// TwinCAT 3 PLC project Untitled1
// ProgramVersion: 3.1.4023.0
// libraries:
//   Tc2_Standard, * (Beckhoff Automation GmbH)
//   Tc2_System, * (Beckhoff Automation GmbH)
//   Tc3_Module, * (Beckhoff Automation GmbH)
// project tree:
//   DataProcessing/QuickSort/ Partition.TcPOU, QuickSort.TcPOU, Swap.TcPOU
//   GVLs/ GVL.TcGVL
//   List/ ListOfINT.TcPOU, NodeINT.TcDUT (not stored)
//   / PlcTask.TcTTO
//   POUs/ ListOfINTTest.TcPOU, MAIN.TcPOU, QuickSortTest.TcPOU
//   Stringify/ Stringify.TcPOU

CONFIGURATION Untitled1
    RESOURCE PLC ON TwinCAT3
        TASK PlcTask(INTERVAL := T#10ms, PRIORITY := 20);
        PROGRAM MAIN WITH PlcTask : MAIN;
    END_RESOURCE
END_CONFIGURATION

// ---- GVLs/GVL.TcGVL
{attribute 'qualified_only'}
VAR_GLOBAL
	vari : int;
END_VAR

// ---- POUs/MAIN.TcPOU

PROGRAM MAIN
VAR
	
END_VAR


ListOfINTTest();

QuickSortTest();

END_PROGRAM

// ---- POUs/ListOfINTTest.TcPOU
PROGRAM ListOfINTTest
VAR
	listOfINTExample : ListOfINT;
	
	// init
	first : BOOL := TRUE;
	reinit : BOOL;
	
	// insert test
	insertTest : BOOL;
	insertNumber : INT := 42;
	insertIndex : INT := 0;
	
	// remove test
	removeTest : BOOL;
	removeIndex : INT := 0;
	
	// prepend test
	prependTest : BOOL;
	prependData : INT := -10;
	
	// removeAll test
	removeAllTest : BOOL;
	
	// debug
	test : ARRAY[0..30] OF INT;
	
	// hokusy pokusy
	info : __SYSTEM.VAR_INFO;
	
END_VAR

IF first THEN
	first := FALSE;
	listOfINTExample.Append(3);
	listOfINTExample.Append(4);
//	listOfINTExample.Append(5).Prepend(2).Prepend(1);
END_IF;
IF reinit THEN
	reinit := FALSE;
	listOfINTExample.FB_init(FALSE, FALSE);
	first := TRUE;
END_IF

IF insertTest THEN
	insertTest := FALSE;
	listOfINTExample.Insert(insertIndex, insertNumber);
END_IF
IF removeTest THEN
	removeTest := FALSE;
	listOfINTExample.Remove(removeIndex);
END_IF
IF removeAllTest THEN
	removeAllTest := FALSE;
	listOfINTExample.RemoveAll();
END_IF


info := __VARINFO(listOfINTExample);
test[0] := listOfINTExample.Get(0);
test[1] := listOfINTExample.Get(1);
test[2] := listOfINTExample.Get(2);
test[3] := listOfINTExample.Get(3);
test[4] := listOfINTExample.Get(4);
test[5] := listOfINTExample.Get(5);
test[6] := listOfINTExample.Get(6);
test[7] := listOfINTExample.Get(7);
test[8] := listOfINTExample.Get(8);
test[9] := listOfINTExample.Get(9);

test[20] := listOfINTExample.Get(-1);
test[21] := listOfINTExample.Get(-2);
test[22] := listOfINTExample.Get(-3);
test[23] := listOfINTExample.Get(-4);
test[24] := listOfINTExample.Get(-5);
test[25] := listOfINTExample.Get(-6);
test[26] := listOfINTExample.Get(-7);
test[27] := listOfINTExample.Get(-8);
test[28] := listOfINTExample.Get(-9);
test[29] := listOfINTExample.Get(-10);

listOfINTExample.count;

END_PROGRAM

// ---- List/ListOfINT.TcPOU

FUNCTION_BLOCK ListOfINT
VAR_INPUT
END_VAR
VAR_OUTPUT
	count : UINT;
END_VAR
VAR
	head : POINTER TO NodeINT := NULL;
	tail : POINTER TO NodeINT := NULL;
END_VAR


// linked list implementation reference:
// https://www.codesdope.com/blog/article/c-linked-lists-in-c-singly-linked-list/


METHOD Append : REFERENCE TO ListOfINT
VAR_INPUT
	data : INT;
END_VAR
VAR
	new : POINTER TO NodeINT;
END_VAR

Append REF= THIS^;

new := __NEW(NodeINT);
new^.data := data;
new^.next := NULL;

IF head = NULL THEN
	head := new;
	tail := new;
ELSE
	tail^.next := new;
	tail := tail^.next;
END_IF
count := count + 1;
END_METHOD


METHOD FB_init : BOOL
VAR_INPUT
	bInitRetains : BOOL; // if TRUE, the retain variables are initialized (warm start / cold start)
	bInCopyCode : BOOL;  // if TRUE, the instance afterwards gets moved into the copy code (online change)
END_VAR
END_METHOD


METHOD Get : INT
VAR_INPUT
	// indexing from end allowed
	// index = 0 returns first element
	// index = 1 returns seconds element
	// index = -1 returns last element
	// index = -2 return before-last element
	index : INT;
END_VAR
VAR
	current : POINTER TO NodeINT := NULL;
	getIndex : INT;
	i : INT;
END_VAR

IF head = NULL THEN
	Get := 0;
	RETURN;
END_IF;

// Return 0 for invalid indexes
IF 	(index >= count) OR	// Indexing from begin begins with 0
	(index < 0 AND index < -count) // Indexing from end begins with -1
THEN
	Get := 0;
	RETURN;
END_IF

getIndex := (count * BOOL_TO_INT(index < 0)) + index - 1;
current := head;
FOR i := 0 TO getIndex DO
	IF current^.next = NULL THEN
		Get := 0; RETURN;
	END_IF
	current := current^.next;
END_FOR
Get := current^.data;
END_METHOD

// Inserts new element into given index. Negative indexing is supported
METHOD Insert : REFERENCE TO ListOfINT
VAR_INPUT
	(*
		0 = Prepend;
		1 = Insert into second position;
		-2 = Insert into second position from end;
		-1 = Append;
	*)
	index : INT;
	data : INT;
END_VAR
VAR
	new : POINTER TO NodeINT;
	current : POINTER TO NodeINT;
	insertIndex : INT;
	i : INT;
END_VAR

Insert REF= THIS^;

new := __NEW(NodeINT);
new^.data := data;

insertIndex := ((count + 1) * BOOL_TO_INT(index < 0)) + index;
NULL;
IF insertIndex >= count // Index too high -> append to end
THEN
	Append(data);
	RETURN;
ELSIF insertIndex <= 0 // Index too high from the end -> prepend to beginning
THEN
	Prepend(data);
	RETURN;
END_IF

current := head;
FOR i := 1 TO insertIndex - 1 DO
	current := current^.next;
END_FOR
new^.next := current^.next;
current^.next := new;
count := count + 1;
END_METHOD


METHOD IsEmpty : BOOL
VAR_INPUT
END_VAR

IsEmpty := head = NULL;
END_METHOD


// Pushes data to the beginning of the list
METHOD Prepend : REFERENCE TO ListOfINT
VAR_INPUT
	data : INT;
END_VAR
VAR
	new : POINTER TO NodeINT;
END_VAR

Prepend REF= THIS^;

new := __NEW(NodeINT);
new^.data := data;
new^.next := head;

IF head = NULL THEN
	head := new;
	tail := new;
ELSE
	head := new;
END_IF
count := count + 1;
END_METHOD


METHOD Remove : REFERENCE TO ListOfINT;
VAR_INPUT
	index : INT;
END_VAR
VAR
	current : POINTER TO NodeINT := NULL;
	removeIndex : INT;	
	nodeToRemove : POINTER TO NodeINT;
	i : INT;
END_VAR

Remove REF= THIS^;

IF head = NULL THEN
	RETURN;
END_IF;

// Cancel removal for invalid indexes
IF 	(index >= count) OR // Indexing from begin begins with 0
	(index < 0 AND index < -count) // Indexing from end begins with -1
THEN
	RETURN;
END_IF

removeIndex := (count * BOOL_TO_INT(index < 0)) + index; 
IF removeIndex = 0 THEN
	nodeToRemove := head;
	head := head^.next;
ELSE
	current := head;
	FOR i := 0 TO removeIndex - 2 DO
		current := current^.next;
	END_FOR
	nodeToRemove := current^.next;
	current^.next := current^.next^.next;
END_IF
IF nodeToRemove = tail THEN
	tail := current;
END_IF
__DELETE(nodeToRemove);
count := count - 1;
END_METHOD

METHOD RemoveAll : REFERENCE TO ListOfINT
VAR_INPUT
END_VAR
WHILE head <> NULL DO
	Remove(0);
END_WHILE
END_METHOD

END_FUNCTION_BLOCK

// ---- POUs/QuickSortTest.TcPOU

PROGRAM QuickSortTest
VAR
	TestArray0 : ARRAY[0..20] OF REAL := [
		1, 2, 3, 4, 5, 6, 7, 8, 9, 10,
		42, 3.14, 0.618, 1.618, 2.618
	];
	TestArray1 : ARRAY[0..1] OF REAL := [0.1, -0.2];
	
	init : BOOL;
	sort : BOOL;
END_VAR


IF init THEN
	init := FALSE;
	reinit();
END_IF

IF sort THEN
	sort := FALSE;
	QuickSort(TestArray0, 0, 20);
	QuickSort(TestArray1, 0, 1);
END_IF


METHOD reinit : BOOL
VAR_INPUT
END_VAR
VAR CONSTANT
	Array0 : ARRAY[0..20] OF REAL := [
		1, 2, 3, 4, 5, 6, 7, 8, 9, 10,
		42, 3.14, 0.618, 1.618, 2.618
	];
	Array1 : ARRAY[0..1] OF REAL := [0.1, -0.2];
END_VAR

TestArray0 := Array0;
TestArray1 := Array1;
END_METHOD

END_PROGRAM

// ---- DataProcessing/QuickSort/QuickSort.TcPOU

// Will sort array of REAL using QuickSort algorythm
FUNCTION QuickSort
VAR_IN_OUT
	ArrayOfREALToSort	: ARRAY[*] OF REAL; // Array to sort
END_VAR
VAR_INPUT
	FirstIndex			: INT; // Start index
	LastIndex			: INT; // End index
END_VAR
VAR 
	PivotLocation		: INT; // Partitioning point
END_VAR


IF FirstIndex < LastIndex THEN
	PivotLocation := Partition(ArrayOfREALToSort, FirstIndex, LastIndex);
	QuickSort(ArrayOfREALToSort, FirstIndex, PivotLocation - 1);
	QuickSort(ArrayOfREALToSort, PivotLocation + 1, LastIndex);
END_IF

END_FUNCTION

// ---- DataProcessing/QuickSort/Partition.TcPOU

// Function used in QuickSort
FUNCTION Partition : INT
VAR_IN_OUT
	ArrayOfREAL			: ARRAY[*] OF REAL; // Partition this array from index nLow to index nHigh
END_VAR
VAR_INPUT
	FirstIndex			: INT; // Starting comparision index
	LastIndex			: INT; // Ending comparision index
END_VAR
VAR
	Pivot				: REAL; // Compared number
	Leftwall			: INT; // New pivot location
	Iterator			: INT; // For iterator variable
END_VAR


Pivot := ArrayOfREAL[LastIndex];
Leftwall := FirstIndex;

FOR Iterator := FirstIndex TO LastIndex - 1 DO
	IF ArrayOfREAL[Iterator] <= Pivot THEN
		Swap(ArrayOfREAL[Iterator], ArrayOfREAL[Leftwall]);
		Leftwall := Leftwall + 1;
	END_IF
END_FOR

Swap(ArrayOfREAL[Leftwall], ArrayOfREAL[LastIndex]);

Partition := Leftwall;

END_FUNCTION

// ---- DataProcessing/QuickSort/Swap.TcPOU

// Swaps values of to variables
FUNCTION Swap
VAR_IN_OUT
	Number1		: REAL;
	Number2		: REAL;
END_VAR
VAR
	Temp		: REAL;
END_VAR


// Just swap pointers
Temp := Number1;
Number1 := Number2;
Number2 := Temp;

END_FUNCTION

// ---- Stringify/Stringify.TcPOU
FUNCTION Stringify : STRING
VAR_INPUT
	info : __SYSTEM.VAR_INFO;
//	another : INT;
END_VAR
VAR
//	info : __SYSTEM.VAR_INFO;
END_VAR

//info := __VARINFO(data);
Stringify := info.Symbol;

END_FUNCTION
